FUNCTION F_PumpStationTurboPumpInterlock : BOOL
VAR_INPUT
END_VAR
VAR
END_VAR

F_PumpStationTurboPumpInterlock := F_CompareGauge(eCompOp:= E_GaugeCompOp._LTE, fReading:=
										GVL_BTS_VAC.fb_PP_GPI_1.PG.rPRESS, 
										eState:= 0, 
										fExpReading:= PTM_INTERLOCK_SP, 
										eExpState:= 0)
									AND F_CompareGauge(eCompOp:= E_GaugeCompOp._LTE, fReading:=
										GVL_BTS_VAC.fb_PP_GPI_2.PG.rPRESS, 
										eState:= 0, 
										fExpReading:= PTM_INTERLOCK_SP, 
										eExpState:= 0)
									AND GVL_BTS_VAC.fb_PP_VVC.M_IsClosed()
									AND GVL_BTS_VAC.fb_PP_PMF.q_stPump.eState = E_PumpState.pumpRUNNING;

END_FUNCTION

(* stored: Version 1.1.0.1, ProductVersion 3.1.4024.0
   POU F_PumpStationTurboPumpInterlock: Id {450d1af3-fb15-4d29-896d-c5cf8ae3a359}, SpecialFunc None *)
